// TwinCAT 3 PLC project MainPLC
// ProgramVersion: 3.1.4024.0
// libraries:
//   Tc2_Standard, * (Beckhoff Automation GmbH)
//   Tc2_System, * (Beckhoff Automation GmbH)
//   Tc3_Module, * (Beckhoff Automation GmbH)
// project tree:
//   / PlcTask.TcTTO
//   POUs/ FB_TrafficLight.TcPOU, MAIN.TcPOU
// real-time tasks:
//   TASK PlcTask: cycle T#10ms, priority 20, ADS port 350

CONFIGURATION MainPLC
    RESOURCE PLC ON TwinCAT3
        TASK PlcTask(INTERVAL := T#10ms, PRIORITY := 20);
        PROGRAM MAIN WITH PlcTask : MAIN;
    END_RESOURCE
END_CONFIGURATION

// ---- POUs/MAIN.TcPOU
PROGRAM MAIN
VAR
	Traffic : FB_TrafficLight;
END_VAR

Traffic();

END_PROGRAM

// ---- POUs/FB_TrafficLight.TcPOU
FUNCTION_BLOCK FB_TrafficLight
VAR_INPUT
END_VAR
VAR_OUTPUT
END_VAR
VAR
	State : INT := 0;
	Timer1 : TON;
	
	Red : BOOL;
	Yellow : BOOL;
	Green : BOOL;
END_VAR

CASE State OF
0:
	Red := TRUE;
	Yellow := FALSE;
	Green := FALSE;
	
	Timer1(IN := TRUE, PT := T#5S);
	IF Timer1.Q THEN
		Timer1(IN := FALSE);
		State := 1;
	END_IF
	
1:
	Red := FALSE;
	Yellow := TRUE;
	Green := FALSE;
	
	Timer1(IN := TRUE, PT := T#5S);
	IF Timer1.Q THEN
		Timer1(IN := FALSE);
		State := 2;
	END_IF
	
2:
	Red := FALSE;
	Yellow := FALSE;
	Green := TRUE;
	
	Timer1(IN := TRUE, PT := T#2S);
	IF Timer1.Q THEN
		Timer1(IN := FALSE);
		State := 0;
	END_IF
	
END_CASE

END_FUNCTION_BLOCK
